Staubli VAL3: getPoint.pgx

public program getPoint(point& x_pPoint[], bool x_bCycle, num x_nIndex)
  local string l_sItem
begin
  // take
  if x_bCycle
    x_pPoint=pt:tTraj[sTrajCycle].tData[x_nIndex].pPoint
  else
    // give back the point
    x_pPoint=pEditPoint.tData[x_nIndex].pPoint
  endIf
end
